{attribute addProperty BoxType "EL2642-0000-0016"}
{attribute addProperty Id "Outputs_Group_1AT %Q*Outputs_Group_E6FE5E20162"}
{attribute addProperty CRC "3804739930"}
{attribute addProperty SizeInBites "16"}
{attribute addProperty SizeInBytes "2"}
TYPE DO_Group_1_Outputs_E2C7B95A :
STRUCT
	{attribute addProperty Name "Outputs_Group_1"}
	Outputs_Group_1 AT %Q* : Outputs_Group_E6FE5E20;
END_STRUCT
END_TYPE

(* stored: Version 1.2.0.0, ProductVersion 3.1.4024.9
   DUT DO_Group_1_Outputs_E2C7B95A: Id {8430a55b-c8b8-47f6-b1db-13f2b621c486} *)
